FUNCTION_BLOCK FB_CommandChangeMaintenance EXTENDS FB_CommandChange IMPLEMENTS ITF_CommandChange
VAR

END_VAR

METHOD Execute : BOOL
VAR_INPUT
END_VAR
END_METHOD

METHOD FB_init : BOOL
VAR_INPUT
	bInitRetains : BOOL; // if TRUE, the retain variables are initialized (warm start / cold start)
	bInCopyCode : BOOL;  // if TRUE, the instance afterwards gets moved into the copy code (online change)
END_VAR
THIS^.SetText (eLocation := E_BaseLocation.pl, wsDescription := "Command change mode - Maintenance");
THIS^.SetText (eLocation := E_BaseLocation.en, wsDescription := "Command change mode - Maintenance");
THIS^.SetText (eLocation := E_BaseLocation.de, wsDescription := "Command change mode - Maintenance");
THIS^.SetName (stName := THIS^.GetTexts ());
END_METHOD

END_FUNCTION_BLOCK

(* stored: Version 1.1.0.1
   POU FB_CommandChangeMaintenance: Id {c8b43683-8473-058f-31ea-a19af17c138c}, SpecialFunc None
   Method Execute: Id {373b072b-e20c-0366-3155-303f3681947e}
   Method FB_init: Id {b905cf72-36fd-02d3-0dd3-6197ba440be8} *)
